// TwinCAT 3 PLC project PLC1
// ProgramVersion: 3.1.4024.0
// libraries:
//   Tc2_Standard, * (Beckhoff Automation GmbH)
//   Tc2_System, * (Beckhoff Automation GmbH)
//   Tc2_Utilities, * (Beckhoff Automation GmbH)
//   Tc3_JsonXml, * (Beckhoff Automation GmbH)
//   Tc3_Module, * (Beckhoff Automation GmbH)
// project tree:
//   HmiUpDateSi2023/1_HmiFunctions/1_Mapping/DUTs/ ST_HmiMapping.TcDUT
//   HmiUpDateSi2023/1_HmiFunctions/1_Mapping/ HmiMapping.TcPOU
//   HmiUpDateSi2023/1_HmiFunctions/2_Add/Class/DUTs/ ST_HmiAdditionData.TcDUT
//   HmiUpDateSi2023/1_HmiFunctions/2_Add/Class/ FB_HmiAddition.TcPOU, I_HmiAddition.TcIO
//   HmiUpDateSi2023/1_HmiFunctions/2_Add/ HmiFunctionAddition.TcPOU
//   HmiUpDateSi2023/1_HmiFunctions/3_Lizenz/Class/ CD_License.TcCD (not stored), GetTc3Licenses.TcPOU, I_GetTc3Licenses.TcIO
//   HmiUpDateSi2023/1_HmiFunctions/3_Lizenz/Class/DUTs/ E_LicenseType.TcDUT, ST_AllLicensesInfos.TcDUT, ST_LicenseDetails.TcDUT, ST_LicenseDetailsSmall.TcDUT, T_JsonDocLicenseInfoSmall.TcDUT
//   HmiUpDateSi2023/1_HmiFunctions/3_Lizenz/ HmiFunctionLizenz.TcPOU
//   / PlcTask.TcTTO
//   POUs/ MAIN.TcPOU
// real-time tasks:
//   TASK PlcTask: cycle T#10ms, priority 20, ADS port 350

CONFIGURATION PLC1
    RESOURCE PLC ON TwinCAT3
        TASK PlcTask(INTERVAL := T#10ms, PRIORITY := 20);
        PROGRAM MAIN WITH PlcTask : MAIN;
    END_RESOURCE
END_CONFIGURATION

// ---- HmiUpDateSi2023/1_HmiFunctions/1_Mapping/DUTs/ST_HmiMapping.TcDUT
TYPE ST_HmiMapping :
STRUCT
    bStart : BOOL;
    bStop: BOOL;
    nValue : INT;
    sBmk : STRING;
END_STRUCT
END_TYPE

// ---- HmiUpDateSi2023/1_HmiFunctions/2_Add/Class/DUTs/ST_HmiAdditionData.TcDUT
TYPE ST_HmiAdditionData :
STRUCT
    ValueA : UDINT;
    ValueB : UDINT;
    Result : UDINT;
END_STRUCT
END_TYPE

// ---- HmiUpDateSi2023/1_HmiFunctions/3_Lizenz/Class/DUTs/E_LicenseType.TcDUT
{attribute 'qualified_only'}
{attribute 'strict'}
TYPE E_LicenseType :
(
    NoType := 0,
    ValidLicenses,
    PendingLicenses,
    DemoLicenses,
    OemLicenses,
    FailedLicenses,
    InvalidLicenses
);
END_TYPE

// ---- HmiUpDateSi2023/1_HmiFunctions/3_Lizenz/Class/DUTs/ST_AllLicensesInfos.TcDUT
TYPE ST_AllLicensesInfos :
STRUCT
    
    ValidLicenses   : ST_LicenseDetails;
    PendingLicenses : ST_LicenseDetails;
    DemoLicenses    : ST_LicenseDetails;
    OemLicenses     : ST_LicenseDetails;
    FailedLicenses  : ST_LicenseDetails;
    InvalidLicenses : ST_LicenseDetails;
    
END_STRUCT
END_TYPE

// ---- HmiUpDateSi2023/1_HmiFunctions/3_Lizenz/Class/DUTs/ST_LicenseDetails.TcDUT
TYPE ST_LicenseDetails :
STRUCT
    Count : UDINT;
    Info : ARRAY[1..Tc2_Utilities.nMaxLicenses] OF ST_TcOnlineLicenseInfoDataEx; // Tc2_Utilities.nMaxLicenses
END_STRUCT
END_TYPE

// ---- HmiUpDateSi2023/1_HmiFunctions/3_Lizenz/Class/DUTs/ST_LicenseDetailsSmall.TcDUT
TYPE ST_LicenseDetailsSmall :
STRUCT
    Count : UDINT;
    Info : ARRAY[1..10] OF ST_TcOnlineLicenseInfoDataEx; // Tc2_Utilities.nMaxLicenses
END_STRUCT
END_TYPE

// ---- HmiUpDateSi2023/1_HmiFunctions/3_Lizenz/Class/DUTs/T_JsonDocLicenseInfoSmall.TcDUT
TYPE T_JsonDocLicenseInfoSmall : STRING(30_000); END_TYPE

// ---- HmiUpDateSi2023/1_HmiFunctions/2_Add/Class/I_HmiAddition.TcIO
INTERFACE I_HmiAddition

{attribute 'TcRpcEnable'}
METHOD AdditionValues : UDINT
VAR_INPUT
    nValueA : UDINT;
    nValueB : UDINT;
END_VAR
END_METHOD

{attribute 'TcRpcEnable'}
METHOD AdditionWithProperty : UDINT
VAR_INPUT
END_VAR
END_METHOD

{attribute 'monitoring' := 'call'}
PROPERTY Result : UDINT
GET
END_GET
END_PROPERTY

{attribute 'monitoring' := 'call'}
PROPERTY ValueA : UDINT
GET
END_GET
SET
END_SET
END_PROPERTY

{attribute 'monitoring' := 'call'}
PROPERTY ValueB : UDINT
GET
END_GET
SET
END_SET
END_PROPERTY

END_INTERFACE

// ---- HmiUpDateSi2023/1_HmiFunctions/3_Lizenz/Class/I_GetTc3Licenses.TcIO
INTERFACE I_GetTc3Licenses

{attribute 'monitoring' := 'call'}
PROPERTY CountDemoLicenses : UDINT
GET
END_GET
END_PROPERTY

{attribute 'monitoring' := 'call'}
PROPERTY CountFailedLicenses : UDINT
GET
END_GET
END_PROPERTY

{attribute 'monitoring' := 'call'}
PROPERTY CountInvalidLicenses : UDINT
GET
END_GET
END_PROPERTY

{attribute 'monitoring' := 'call'}
PROPERTY CountOemLicenses : UDINT
GET
END_GET
END_PROPERTY

{attribute 'monitoring' := 'call'}
PROPERTY CountPendingLicenses : UDINT
GET
END_GET
END_PROPERTY

{attribute 'monitoring' := 'call'}
PROPERTY CountValidLicenses : UDINT
GET
END_GET
END_PROPERTY

{attribute 'TcRpcEnable'}
METHOD GetJsonDataLicenses : T_JsonDocLicenseInfoSmall
VAR_INPUT
    LicensesType : UINT; //E_LicenseType;
END_VAR
END_METHOD

{attribute 'monitoring' := 'call'}
PROPERTY JsonDataDemoLicenses : T_JsonDocLicenseInfoSmall
GET
END_GET
END_PROPERTY

{attribute 'monitoring' := 'call'}
PROPERTY JsonDataFailedLicenses : T_JsonDocLicenseInfoSmall
GET
END_GET
END_PROPERTY

{attribute 'monitoring' := 'call'}
PROPERTY JsonDataInvalidLicenses : T_JsonDocLicenseInfoSmall
GET
END_GET
END_PROPERTY

{attribute 'monitoring' := 'call'}
PROPERTY JsonDataOemLicenses : T_JsonDocLicenseInfoSmall
GET
END_GET
END_PROPERTY

{attribute 'monitoring' := 'call'}
PROPERTY JsonDataPendingLicenses : T_JsonDocLicenseInfoSmall
GET
END_GET
END_PROPERTY

{attribute 'monitoring' := 'call'}
PROPERTY JsonDataValidLicenses : T_JsonDocLicenseInfoSmall
GET
END_GET
END_PROPERTY

END_INTERFACE

// ---- POUs/MAIN.TcPOU
PROGRAM MAIN
VAR
END_VAR


// PLC Methode
 HmiMapping();
 HmiFunctionAddition();
 HmiFunctionLizenz();

// Hmi Classic

// Hmi Vue3

// Testing

END_PROGRAM

// ---- HmiUpDateSi2023/1_HmiFunctions/1_Mapping/HmiMapping.TcPOU
PROGRAM HmiMapping
VAR
    nNoAutoMapping : INT := 1;
    
    {attribute 'TcHmiSymbol.AddSymbol'}
    nAutoMapping : INT := 2;

    {attribute 'TcHmiSymbol.AddSymbol'}
    {attribute 'TcHmiSymbol.ReadOnly'}
    nAutoMappingReadOnly : INT := 3;

    {attribute 'TcHmiSymbol.AddSymbol'}
    {attribute 'TcHmiSymbol.AddSymbol.Hidden'}
    nAutoMappingHidden : INT := 4;

    {attribute 'TcHmiSymbol.AddSymbol'}
    {attribute 'TcHmiSymbol.AddSymbol.UserGroups' := 'GroupWorkshop'}
    nAutoMappingUserGroup : INT := 5;
    
    {attribute 'TcHmiSymbol.AddSymbol'}
    stAutoMapping : ST_HmiMapping := (sBmk :='AutoMapping', nValue := 20, bStart := TRUE);

END_VAR

END_PROGRAM

// ---- HmiUpDateSi2023/1_HmiFunctions/2_Add/HmiFunctionAddition.TcPOU
PROGRAM HmiFunctionAddition
VAR
    // Instanz
    fbHmiAddition : FB_HmiAddition;

    // Interface
    iHmiAddition : I_HmiAddition := fbHmiAddition;

    // Addition Data
    stHmiAdditionData : ST_HmiAdditionData;

    // Test
    bTestAdditionProperties : BOOL;    
    bTestAdditionValue : BOOL;    

END_VAR



IF bTestAdditionProperties THEN
    bTestAdditionProperties := FALSE;
    // set Properties
    iHmiAddition.ValueA := stHmiAdditionData.ValueA;
    iHmiAddition.ValueB := stHmiAdditionData.ValueB;
    
    // call
    iHmiAddition.AdditionWithProperty();
    
    // Result
    stHmiAdditionData.Result := iHmiAddition.Result; 
END_IF


IF bTestAdditionValue THEN
    bTestAdditionValue := FALSE;
    stHmiAdditionData.Result := iHmiAddition.AdditionValues(stHmiAdditionData.ValueA, stHmiAdditionData.ValueB);   
END_IF

END_PROGRAM

// ---- HmiUpDateSi2023/1_HmiFunctions/2_Add/Class/FB_HmiAddition.TcPOU
{attribute 'TcRpcEnable'}
FUNCTION_BLOCK PUBLIC FB_HmiAddition IMPLEMENTS I_HmiAddition
VAR_INPUT
END_VAR
VAR_OUTPUT
END_VAR
VAR
    _HmiData : ST_HmiAdditionData;
END_VAR

METHOD PRIVATE Addition : UDINT
VAR_INPUT
	nValueA	: UDINT;
	nValueB	: UDINT;
END_VAR
 Addition := nValueA + nValueB;
END_METHOD

{attribute 'TcRpcEnable'}
METHOD AdditionValues : UDINT
VAR_INPUT
	nValueA	: UDINT;
	nValueB	: UDINT;
END_VAR
VAR
    nReturn : UDINT;
END_VAR

 // set property
 ValueA := nValueA;
 ValueB := nValueB;

 // call method
 nReturn := Addition(nValueA, nValueB);
 
 // set Result
 _HmiData.Result := nReturn;
 
 // return
 AdditionValues := nReturn;
END_METHOD

{attribute 'TcRpcEnable'}
METHOD PUBLIC AdditionWithProperty : UDINT
VAR_INPUT
END_VAR
VAR
    nReturn : UDINT;
END_VAR

 // call method
 nReturn := Addition(ValueA, ValueB);
 
 // set Result
 _HmiData.Result := nReturn;
 
 // return
 AdditionWithProperty := nReturn;
END_METHOD

{attribute 'monitoring' := 'call'}
PROPERTY Result : UDINT
GET

Result := _HmiData.Result;
END_GET
END_PROPERTY

{attribute 'monitoring' := 'call'}
PROPERTY ValueA : UDINT
GET

ValueA := _HmiData.ValueA;
END_GET
SET

_HmiData.ValueA := ValueA;
END_SET
END_PROPERTY

{attribute 'monitoring' := 'call'}
PROPERTY ValueB : UDINT
GET

ValueB := _HmiData.ValueB;
END_GET
SET

_HmiData.ValueB := ValueB;
END_SET
END_PROPERTY

END_FUNCTION_BLOCK

// ---- HmiUpDateSi2023/1_HmiFunctions/3_Lizenz/HmiFunctionLizenz.TcPOU
PROGRAM HmiFunctionLizenz
VAR
    fbAllLicenses : GetTc3Licenses(NetId := '');
    iAllLicenses : I_GetTc3Licenses := fbAllLicenses;
    bExecute : BOOL := TRUE;

    bGenerateJsonData : BOOL;
    sJsonDoc      : T_JsonDocLicenseInfoSmall;
    nCountLicense : UDINT;
    nType : UINT := 3; // Demo
    
END_VAR


fbAllLicenses.GetAllLicenses(bExecute);

IF bGenerateJsonData THEN
    bGenerateJsonData := FALSE;
//    sJsonDoc := fbAllLicenses.JsonDataDemoLicenses;
    sJsonDoc := iAllLicenses.GetJsonDataLicenses(nType);
    nCountLicense := fbAllLicenses.CountDemoLicenses;  
END_IF

END_PROGRAM

// ---- HmiUpDateSi2023/1_HmiFunctions/3_Lizenz/Class/GetTc3Licenses.TcPOU
{attribute 'TcRpcEnable'}
FUNCTION_BLOCK GetTc3Licenses IMPLEMENTS I_GetTc3Licenses
VAR_INPUT
END_VAR
VAR_OUTPUT
END_VAR
VAR
END_VAR
VAR
    // Internal
    fbGetLicensesEx : FB_GetLicensesEx;
    stAllLicensesInfos : ST_AllLicensesInfos;
    
    _sNetId   : T_AmsNetId;
    
    _fbJson         : FB_JsonSaxWriter;
    _fbJsonDataType : FB_JsonReadWriteDataType;
    
END_VAR
VAR
    stInfoData : ST_LicenseDetailsSmall;
    sReturn : STRING(30_000);
END_VAR


// include: Tc2_Utilities
// Realtime -> Global Max Stack = 2048kb

{attribute 'monitoring' := 'call'}
PROPERTY CountDemoLicenses : UDINT
GET

CountDemoLicenses := stAllLicensesInfos.DemoLicenses.Count;
END_GET
END_PROPERTY

{attribute 'monitoring' := 'call'}
PROPERTY CountFailedLicenses : UDINT
GET

CountFailedLicenses := stAllLicensesInfos.FailedLicenses.Count;
END_GET
END_PROPERTY

{attribute 'monitoring' := 'call'}
PROPERTY CountInvalidLicenses : UDINT
GET

CountInvalidLicenses := stAllLicensesInfos.InvalidLicenses.Count;
END_GET
END_PROPERTY

{attribute 'monitoring' := 'call'}
PROPERTY CountOemLicenses : UDINT
GET

CountOemLicenses := stAllLicensesInfos.OemLicenses.Count;
END_GET
END_PROPERTY

{attribute 'monitoring' := 'call'}
PROPERTY CountPendingLicenses : UDINT
GET

CountPendingLicenses := stAllLicensesInfos.PendingLicenses.Count;
END_GET
END_PROPERTY

{attribute 'monitoring' := 'call'}
PROPERTY CountValidLicenses : UDINT
GET

CountValidLicenses := stAllLicensesInfos.ValidLicenses.Count;
END_GET
END_PROPERTY

METHOD FB_init : BOOL
VAR_INPUT
	bInitRetains : BOOL; // if TRUE, the retain variables are initialized (warm start / cold start)
	bInCopyCode : BOOL;  // if TRUE, the instance afterwards gets moved into the copy code (online change)
    NetId   : T_AmsNetId;
END_VAR

_sNetId := NetId;
END_METHOD

METHOD PUBLIC GetAllLicenses : HRESULT
VAR_INPUT
    bExecute : REFERENCE to BOOL;
END_VAR

IF bExecute THEN
    fbGetLicensesEx(
        bExecute:= bExecute, 
        tTimeout:= , 
        sNetId:= _sNetId, 
        bBusy=> , 
        bError=> , 
        nErrorId=> , 
        nValidLicenses=> stAllLicensesInfos.ValidLicenses.Count, 
        aValidLicenses=> stAllLicensesInfos.ValidLicenses.Info, 
        nPendingLicenses=> stAllLicensesInfos.PendingLicenses.Count, 
        aPendingLicenses=> stAllLicensesInfos.PendingLicenses.Info, 
        nDemoLicenses=> stAllLicensesInfos.DemoLicenses.Count, 
        aDemoLicenses=> stAllLicensesInfos.DemoLicenses.Info, 
        nOemLicenses=> stAllLicensesInfos.OemLicenses.Count, 
        aOemLicenses=> stAllLicensesInfos.OemLicenses.Info, 
        nFailedLicenses=> stAllLicensesInfos.FailedLicenses.Count, 
        aFailedLicenses=> stAllLicensesInfos.FailedLicenses.Info, 
        nInvalidLicenses=> stAllLicensesInfos.InvalidLicenses.Count, 
        aInvalidLicenses=> stAllLicensesInfos.InvalidLicenses.Info);
    
    IF NOT fbGetLicensesEx.bBusy THEN
        bExecute := FALSE;
	END_IF
END_IF
END_METHOD

{attribute 'TcRpcEnable'}
METHOD GetJsonDataLicenses : T_JsonDocLicenseInfoSmall
VAR_INPUT
	LicensesType	: UINT; //E_LicenseType;
END_VAR

CASE LicensesType OF
    E_LicenseType.NoType:
        GetJsonDataLicenses := '';
    E_LicenseType.ValidLicenses:
        GetJsonDataLicenses := JsonDataValidLicenses;
    E_LicenseType.PendingLicenses:
        GetJsonDataLicenses := JsonDataPendingLicenses;
    E_LicenseType.DemoLicenses:
        GetJsonDataLicenses := JsonDataDemoLicenses;
    E_LicenseType.OemLicenses:
        GetJsonDataLicenses := JsonDataOemLicenses;
    E_LicenseType.FailedLicenses:
        GetJsonDataLicenses := JsonDataFailedLicenses;
    E_LicenseType.InvalidLicenses:
        GetJsonDataLicenses := JsonDataInvalidLicenses;
END_CASE
END_METHOD

METHOD PRIVATE GetJsonLicenseDetailSmall : HRESULT
VAR_INPUT
    AdrLicense : XWORD;
    refJsonDoc : REFERENCE TO STRING(30_000);
END_VAR

//Tc2_System.MEMCPY(ADR(stInfoData), ADR(stAllLicensesInfos.ValidLicenses), SIZEOF(stInfoData));
Tc2_System.MEMCPY(ADR(stInfoData), AdrLicense, SIZEOF(stInfoData));

_fbJson.ResetDocument();
_fbJsonDataType.AddJsonValueFromSymbol(_fbJson, 'ST_LicenseDetailsSmall', SIZEOF(stInfoData), ADR(stInfoData));
_fbJson.CopyDocument(sReturn, SIZEOF(sReturn));

refJsonDoc := sReturn;

GetJsonLicenseDetailSmall := S_OK;
END_METHOD

{attribute 'monitoring' := 'call'}
PROPERTY JsonDataDemoLicenses : T_JsonDocLicenseInfoSmall
GET

GetJsonLicenseDetailSmall(ADR(stAllLicensesInfos.DemoLicenses), JsonDataDemoLicenses);
END_GET
END_PROPERTY

{attribute 'monitoring' := 'call'}
PROPERTY JsonDataFailedLicenses : T_JsonDocLicenseInfoSmall
GET

GetJsonLicenseDetailSmall(ADR(stAllLicensesInfos.FailedLicenses), JsonDataFailedLicenses);
END_GET
END_PROPERTY

{attribute 'monitoring' := 'call'}
PROPERTY JsonDataInvalidLicenses : T_JsonDocLicenseInfoSmall
GET

GetJsonLicenseDetailSmall(ADR(stAllLicensesInfos.InvalidLicenses), JsonDataInvalidLicenses);
END_GET
END_PROPERTY

{attribute 'monitoring' := 'call'}
PROPERTY JsonDataOemLicenses : T_JsonDocLicenseInfoSmall
GET

GetJsonLicenseDetailSmall(ADR(stAllLicensesInfos.OemLicenses), JsonDataOemLicenses);
END_GET
END_PROPERTY

{attribute 'monitoring' := 'call'}
PROPERTY JsonDataPendingLicenses : T_JsonDocLicenseInfoSmall
GET

GetJsonLicenseDetailSmall(ADR(stAllLicensesInfos.PendingLicenses), JsonDataPendingLicenses);
END_GET
END_PROPERTY

{attribute 'monitoring' := 'call'}
PROPERTY JsonDataValidLicenses : T_JsonDocLicenseInfoSmall
GET

GetJsonLicenseDetailSmall(ADR(stAllLicensesInfos.ValidLicenses), JsonDataValidLicenses);
END_GET
END_PROPERTY

END_FUNCTION_BLOCK
